// TIA Portal V18 export
TYPE "LGasp_TypeERP_packet"
// stored: IsFailsafeCompliant false
   STRUCT
      CastingCode : String[30];   // Codice colata (dal cliente)
      LogisticID : String[30];   // ID Logistico (dal cliente)
      ProfileCode : String[30];   // Codice profilo
      MaterialCode : String[30];   // Materiale
      SteelGrade : String[30];   // TIpo acciaio
      Length : Real;   // [mm] Lunghezza pezzi su pacco
      Width : Real;   // [mm] Larghezza pezzi su pacco
      Height : Real;   // [mm] Altezza pezzi su pacco
      Thickness : Real;   // [mm] Spessore lamiera
      Aletta : Real;   // [mm] Aletta pezzi su pacco
      Weight_Tot : Real;   // [kg] Peso totale pacco
      Qty_Tot : Int;   // Quantità pezzi
      collo : Int;   // identificatico pacco 210100085
      workorder : DInt;   // dato 210100085
      IDERP : DInt;   // dato 210100085
      paccoparziale { ExternalAccessible := 'False'; ExternalVisible := 'False'; ExternalWritable := 'False'} : Bool;   // pacco non completato 210100085
   END_STRUCT;
END_TYPE
